KUKA KRL program: LeafMillKey.src, LeafMillKey.dat

--- LeafMillKey.src ---
&ACCESS RVEO
&REL 2
DEF LeafMillKey(stKey:IN,eProfile:IN)
   ;FOLD DECL
      DECL ST_Dim3 stKey
      DECL E_ProfileType eProfile
      DECL POS xKey,xAwayKey,xAboveAwayKey,xAboveTable
      DECL POS xWall[4],xAboveWall[4],xInsideWall[4],xCutPath[4,12]
      DECL INT iWall,iPoint,iPointFinish
   ;ENDFOLD (DECL)
   ;FOLD INI
      ;FOLD BASISTECH INI
         GLOBAL INTERRUPT DECL 3 WHEN $STOPMESS==TRUE DO IR_STOPM ( )
         INTERRUPT ON 3
         BAS (#INITMOV,0 )
      ;ENDFOLD (BASISTECH INI)
      ;FOLD USER INI
         xKey = xOriIni
         xKey.x = stKey.rX
         xKey.y = ProfileWallDist(eProfile,#Y,1)
         xKey.z = stKey.rZ

         xAwayKey = xAwayKeyOffset:xKey
         xAboveAwayKey = xAboveKeyOffset:xAwayKey
         xAboveTable = xAboveTableOffset:xAwayKey

         FOR iWall=1 TO iWallSize STEP 1
            xWall[iWall] = xKey
            xWall[iWall].y = ProfileWallDist(eProfile,#Y,iWall)
            xAboveWall[iWall] = xWall[iWall]:xAboveWallOffset
            xInsideWall[iWall] = xWall[iWall]:xInsideWallOffset

            FOR iPoint=1 TO 6 STEP 1
               xCutPath[iWall,iPoint] = xWall[iWall]:GetRectangleOffset(stKeyRoughDim,iPoint)
               xCutPath[iWall,iPoint].y = xWall[iWall].y - ABS(xInsideWallOffset.z)
               iPointFinish = iPoint + 6
               xCutPath[iWall,iPointFinish] = xWall[iWall]:GetRectangleOffset(stKeyFinishDim[iWall],iPoint)
               xCutPath[iWall,iPointFinish].y = xWall[iWall].y - ABS(xInsideWallOffset.z)
            ENDFOR
         ENDFOR
      ;ENDFOLD (USER INI)
   ;ENDFOLD (INI)

   BAS(#INITMOV)
   SetBaseTool(#MillTable,#Cutter16)

   SetVel(#SpindleIdle)
   LIN xAboveTable C_DIS
   Spindle(#eRun,#SpindleHITECO,17900)

   SetVel(#SpindleIdle)
   LIN xAboveAwayKey C_DIS
   LIN xAwayKey C_DIS

   FOR iWall=1 TO iWallSize STEP 1
      SetVel(#SpindleIdle)
      LIN xAboveWall[iWall] C_DIS
      SetVel(#MillPuncture)
      LIN xInsideWall[iWall] C_DIS

      SetVel(#MillKey)
      FOR iPoint=1 TO iCutPathSize STEP 1
         LIN xCutPath[iWall,iPoint] C_DIS
      ENDFOR

      SetVel(#SpindleIdle)
      LIN xInsideWall[iWall] C_DIS
   ENDFOR

   SetVel(#SpindleIdle)
   LIN xAwayKey C_DIS
   LIN xAboveAwayKey C_DIS
   LIN xAboveTable

END

DEFFCT POS GetRectangleOffset(stLockDim:IN,iPoint:IN)
   DECL ST_Dim3 stLockDim,stDistFactor,stDist
   DECL POS xOffset
   DECL INT iPoint

   xOffset = $NULLFRAME
   stDist.rX = (stLockDim.rX-grFiCutter16)/2
   stDist.rY = (stLockDim.rY-grFiCutter16)/2

   SWITCH iPoint
      CASE 1
         stDistFactor = {rX  0.0,rY -1.0}
      CASE 2
         stDistFactor = {rX +1.0,rY -1.0}
      CASE 3
         stDistFactor = {rX +1.0,rY +1.0}
      CASE 4
         stDistFactor = {rX -1.0,rY +1.0}
      CASE 5
         stDistFactor = {rX -1.0,rY -1.0}
      CASE 6
         stDistFactor = {rX  0.0,rY -1.0}
      DEFAULT
         HALT
   ENDSWITCH

   xOffset.x = stDistFactor.rX * stDist.rX
   xOffset.y = stDistFactor.rY * stDist.rY

   RETURN xOffset

ENDFCT

--- LeafMillKey.dat ---
&ACCESS RVEO
&REL 2
DEFDAT LeafMillKey
;FOLD EXTERNAL DECLARATIONS;%{PE}%MKUKATPBASIS,%CEXT,%VCOMMON,%P
;FOLD BASISTECH EXT;%{PE}%MKUKATPBASIS,%CEXT,%VEXT,%P
EXT  BAS (BAS_COMMAND  :IN,REAL  :IN )
DECL INT SUCCESS
;ENDFOLD (BASISTECH EXT)
;FOLD USER EXT;%{E}%MKUKATPUSER,%CEXT,%VEXT,%P
;Make here your modifications

;ENDFOLD (USER EXT)
;ENDFOLD (EXTERNAL DECLERATIONS)

DECL CONST POS xOriIni = {x 0,y 0,z 0,a 0,b 0,c -90}

DECL CONST INT iWallSize = 4
DECL CONST INT iCutPathSize = 12

DECL CONST REAL rWallThick = 4.0
DECL CONST REAL rVertMillDistX = 5.0
DECL CONST ST_Dim3 stKeyRoughDim = {rX 35,rY 19}
DECL CONST ST_Dim3 stKeyFinishDim[4]
stKeyFinishDim[1] = {rX 38,rY 22}
stKeyFinishDim[2] = {rX 38,rY 22}
stKeyFinishDim[3] = {rX 37,rY 21}
stKeyFinishDim[4] = {rX 37,rY 21}

DECL CONST POS xAboveTableOffset = {x 0,y 0,z 200,a 0,b 0,c 0}
DECL CONST POS xAwayKeyOffset = {x 0,y 100,z 0,a 0,b 0,c 0}
DECL CONST POS xAboveKeyOffset = {x 0,y 0,z 150,a 0,b 0,c 0}
DECL CONST POS xAboveWallOffset = {x 6,y 0,z 0,a 0,b 0,c 0}
DECL CONST POS xInsideWallOffset = {x -6,y 0,z -6,a 0,b 0,c 0}

ENDDAT
